Universal Robots PolyScope program: pos4.urp

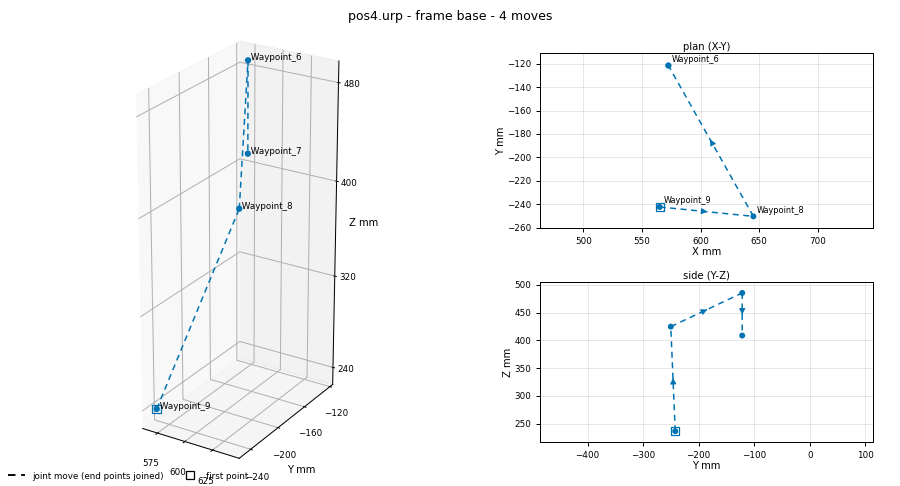
[picture p0: tool path of pos4.urp in frame base, 4 of 4 moves have a stored position in this frame; points joined in program order, loops and branches not executed]
Program pos4 (installation=default directory=/programs/Nicolas_Arteaga/quality createdIn=5.12.4.1101661 lastSavedIn=5.12.4.1101661 robotSerialNumber=20225502378)
Calibrated DH parameters: a=[0.00022, -0.425328, -0.389701, 0.000059, 0.000065, 0]; d=[0.162608, 0.803456, 9.992211, -10.662202, 0.099702, 0.099559]; alpha=[1.570756, 0.001543, 0.004316, 1.570651, -1.570122, 0]; deltaTheta=[0, 0.002917, 0.116094, -0.119008, 0, -0.000001]
Robot Program (runOnlyOnce=true)
  MoveJ speed 60 deg/s, acceleration 80 deg/s^2 (useActiveTCP=true) feature=Base
    Waypoint Waypoint_9: TCP in base x=565.027 y=-242.247 z=236.41 mm, rx=-0.2913 ry=1.6112 rz=0.3439 rad; joints [113.27, -55.479, 94.871, 44.262, 2.977, 188.935] deg; TCP offset x=0 y=0 z=191.5 mm, rx=0 ry=0 rz=0 rad
    Waypoint Waypoint_8: TCP in base x=644.963 y=-250.234 z=424.745 mm, rx=-0.4223 ry=1.4905 rz=0.4378 rad; joints [121.021, -52.336, 61.566, 67.994, -2.525, 192.758] deg
    Waypoint Waypoint_6: TCP in base x=572.488 y=-121.624 z=485.395 mm, rx=-1.4669 ry=0.8076 rz=-0.7838 rad; joints [121.615, -73.605, 85.33, 82.996, 2.356, 84.774] deg; TCP offset x=0 y=0 z=191.5 mm, rx=0 ry=0 rz=0 rad
    Waypoint Waypoint_7: TCP in base x=572.477 y=-121.647 z=408.681 mm, rx=-1.4669 ry=0.8076 rz=-0.7839 rad; joints [121.624, -70.654, 92.721, 71.319, 2.368, 86.105] deg; TCP offset x=0 y=0 z=191.5 mm, rx=0 ry=0 rz=0 rad
    'measure pressure pos2'
